RoboDK station: Program_VDL_Testobject_AMR_mapped_v2.rdk

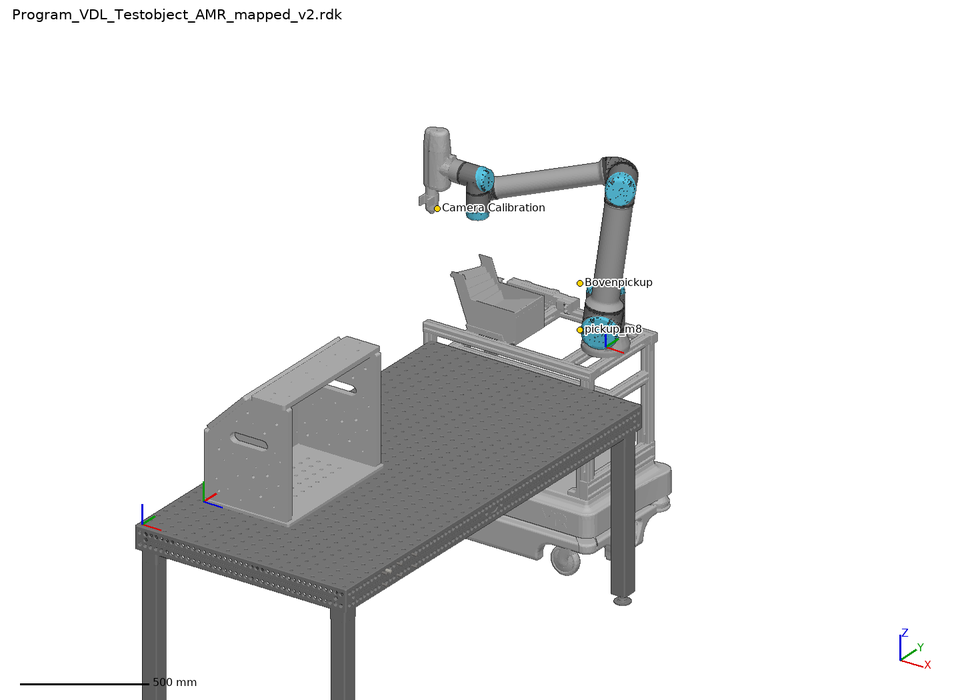
[picture v0: the station drawn from its stored meshes, robots at their saved joint values, targets as dots, program paths as lines]
Station Program_VDL_Testobject_AMR_mapped_v2 (saved by RoboDK 6.0.1). Poses are relative to the parent item; angles as X-Y-Z fixed-axis rotations.
Station parameters (name, value as stored): CollisionFreePlanner, UR10e, CollisionFreePlanner-Rob UR10e, Simplify-Mesh-Settings, Simplify-Mesh-Settings-Backup
  - object Lastafel at (0, 0, 0) mm, size 1021.8 x 2000 x 842 mm
  - object Lastafel_simplified at (0, 0, 0) mm, size 1000 x 2000 x 802.1 mm
  - frame Base frame at (-1000, -100, 50) mm
    - target Camera Calibration (Cartesian target) at (100, 1850, 650) mm, rotated rx 180 ry 0 rz -180 deg; joints [29.689, -97.282, 108.694, 168.588, -119.69, 90.001] of UR10e
  - frame UR10e Base at (-350, 2100, 116.62) mm
    - robot UR10e: 6 axes, payload 10 kg, reach 1300 mm, repeatability 0.05 mm, weight 28.9 kg
        modified DH rows (alpha deg, a mm, theta deg, d mm): 0, 0, 0, 180.7; 90, 0, 180, 0; 0, 612.6, 0, 0; 0, 571.335, 0, 174.15; -90, 0, 0, 119.85; 90, 0, 180, 116.55
        joint limits [-360, -125, -30, -180, -180, -180] to [360, 0, 180, 180, 180, 180]; home [30.872, -95.296, 116.362, -22.187, 121.11, 179.827]; saved at [29.689, -97.282, 108.694, 168.588, -119.69, 90.001]
      - tool Screwdriver, TCP at (210, -1, 100.64) mm, rotated rx 0 ry -90 rz 180 deg, size 98 x 366.6 x 139.7 mm
      - tool Screwdriver simplified, TCP at (210, -1, 100.64) mm, rotated rx 0 ry -90 rz 180 deg, size 98.1 x 366.6 x 139.8 mm
      - tool Camera, TCP at (211.79, -40.21, 100.64) mm, rotated rx 90 ry -90 rz 90 deg
    - object Assembly mir + frame aangepast naar ur10e versie 2 at (-733.08, 277.19, -552.66) mm, rotated rx 90 ry 0 rz 0.45 deg, size 901.1 x 1139.6 x 580.4 mm, geometry from Assembly mir + frame aangepast naar ur10e versie 2.STEP
    - object Mir + frame simplified at (-733.08, 277.19, -552.66) mm, rotated rx 90 ry 0 rz 0.45 deg, size 925.7 x 1139.7 x 582 mm
  - frame CSV Frame at (-919, 200, 49.99) mm, rotated rx 90 ry 0 rz 90.11 deg
    - object Test object at (0, 0.01, 0) mm, size 650 x 517 x 400 mm, geometry from Test object.STEP
    - object Test object simplified at (0, 0.01, 0) mm, size 650.1 x 517 x 436.5 mm
    - target pickup_m8 (joint target) at (1798.98, 166.61, 522.55) mm, rotated rx -90.64 ry -89.89 rz -179.36 deg; joints [-54.773, -65.69, 138.921, 106.769, -35.227, 90] of UR10e
    - target Bovenpickup (joint target) at (1798.98, 366.61, 522.55) mm, rotated rx -90.64 ry -89.89 rz -179.36 deg; joints [-54.773, -102.749, 117.612, -14.864, 35.227, -90] of UR10e
